Omron CX-Programmer project NewProject (CX-Programmer 9.75)

# PLC NewPLC1: CP2E-N N

## Global symbols (name address type ; comment)
W2.00 BOOL  ; ModbusStatus
0.00 BOOL  ; PROXY STOP KONVEYOR
0.01 BOOL  ; PROXY BOWL DISPENSER
0.02 BOOL  ; START BUTTON
100.00 BOOL  ; MOTOR BOWL DISPENSER
100.01 BOOL  ; MOTOR KONVEYOR
100.02 BOOL  ; MOTOR KONVEYOR
100.06 BOOL  ; MOTOR LINEAR ACTUATOR
10.02 BOOL  ; Cup Dispensed
200.00 BOOL  ; RELAY START
200.01 BOOL  ; RELAY START KONVEYOR
200.02 BOOL  ; RELAY ACTUATOR
200.03 BOOL  ; MOTOR BOWL
200.04 BOOL  ; RESET COUNTER
C0 CHANNEL  ; COMPILE MOTOR BOWL
T000 BOOL  ; TIMER ACTUATOR
T001 BOOL  ; TIMER START KONVEYOR
T002 BOOL  ; TIMER START KONVEYOR AFTER BOWL
T003 BOOL  ; START BOWL
W100.01 BOOL  ; MieKering_Ready
W100.02 BOOL  ; Cup_Jalan
W100.03 BOOL  ; RebusMie1_Start
W100.04 BOOL  ; RebusMie1_Done
W100.05 BOOL  ; RebusMie2_Start
W100.06 BOOL  ; RebusMie2_Done
W100.07 BOOL  ; RebusMie3_Start
W100.08 BOOL  ; RebusMie3_Done
W100.09 BOOL  ; Picked Cup
W10.00 BOOL  ; RST
W10.01 BOOL  ; MieKering_Picked
W10.02 BOOL  ; Cup dispensed
W10.03 BOOL  ; CupReady
W11.00 BOOL  ; Delay 1sec Trigger
W12.00 BOOL  ; 1 Sec Delay
W1.00 BOOL  ; MieKering_Arrived
W1.01 BOOL  ; MieKering_Picked
W1.02 BOOL  ; Cup_Dropped
W5.00 BOOL  ; Start MODBUS
FB_MODBUSTCP_SERVER _CP2E003_ExecuteModTcpServer
Order1_Menu D110 CHANNEL
Order1_Topping1 D100 CHANNEL
Order1_Topping2 D101 CHANNEL
Order1_Topping3 D102 CHANNEL
Order2_Menu D111 CHANNEL
Order2_Topping1 D103 CHANNEL
Order2_Topping2 D104 CHANNEL
Order2_Topping3 D105 CHANNEL
Order3_Menu D112 CHANNEL
Order3_Topping1 D106 CHANNEL
Order3_Topping2 D107 CHANNEL
Order3_Topping3 D108 CHANNEL
Start_Order W100.00 BOOL

## Program MODBUS (cyclic task 0)

### Section MODBUS

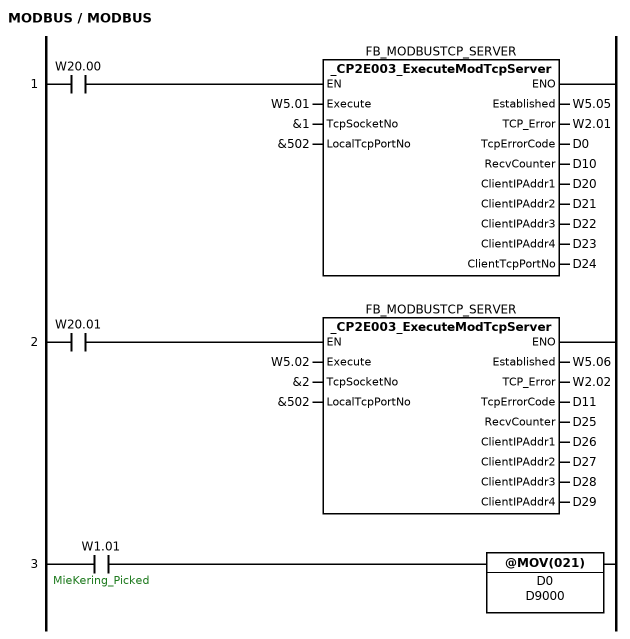
; rung 1
LD W20.00
CALL FB_MODBUSTCP_SERVER : _CP2E003_ExecuteModTcpServer (Execute := W5.01, TcpSocketNo := &1, LocalTcpPortNo := &502, Established => W5.05, TCP_Error => W2.01, TcpErrorCode => D0, RecvCounter => D10, ClientIPAddr1 => D20, ClientIPAddr2 => D21, ClientIPAddr3 => D22, ClientIPAddr4 => D23, ClientTcpPortNo => D24)
; rung 2
LD W20.01
CALL FB_MODBUSTCP_SERVER : _CP2E003_ExecuteModTcpServer (Execute := W5.02, TcpSocketNo := &2, LocalTcpPortNo := &502, Established => W5.06, TCP_Error => W2.02, TcpErrorCode => D11, RecvCounter => D25, ClientIPAddr1 => D26, ClientIPAddr2 => D27, ClientIPAddr3 => D28, ClientIPAddr4 => D29)
; rung 3
LD W1.01  ; MieKering_Picked
@MOV(021) D0 D9000

### Section Main

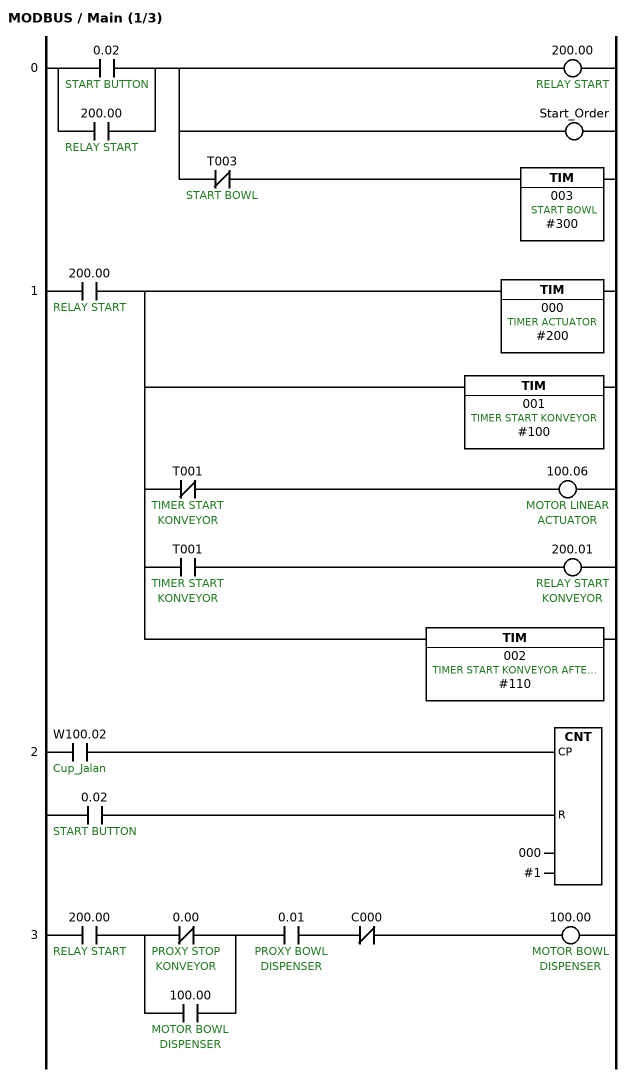
; rung 0
LD 0.02  ; START BUTTON
OR 200.00  ; RELAY START
OUT 200.00  ; RELAY START
OUT Start_Order
ANDNOT T003  ; START BOWL
TIM 003 #300  ; START BOWL
; rung 1
LD 200.00  ; RELAY START
OUT TR0
TIM 000 #200  ; TIMER ACTUATOR
TIM 001 #100  ; TIMER START KONVEYOR
ANDNOT T001  ; TIMER START KONVEYOR
OUT 100.06  ; MOTOR LINEAR ACTUATOR
LD TR0
AND T001  ; TIMER START KONVEYOR
OUT 200.01  ; RELAY START KONVEYOR
LD TR0
TIM 002 #110  ; TIMER START KONVEYOR AFTER BOWL
; rung 2
LD W100.02  ; Cup_Jalan
LD 0.02  ; START BUTTON
CNT 000 #1
; rung 3
LD 200.00  ; RELAY START
LDNOT 0.00  ; PROXY STOP KONVEYOR
OR 100.00  ; MOTOR BOWL DISPENSER
ANDLD
AND 0.01  ; PROXY BOWL DISPENSER
ANDNOT C000
OUT 100.00  ; MOTOR BOWL DISPENSER

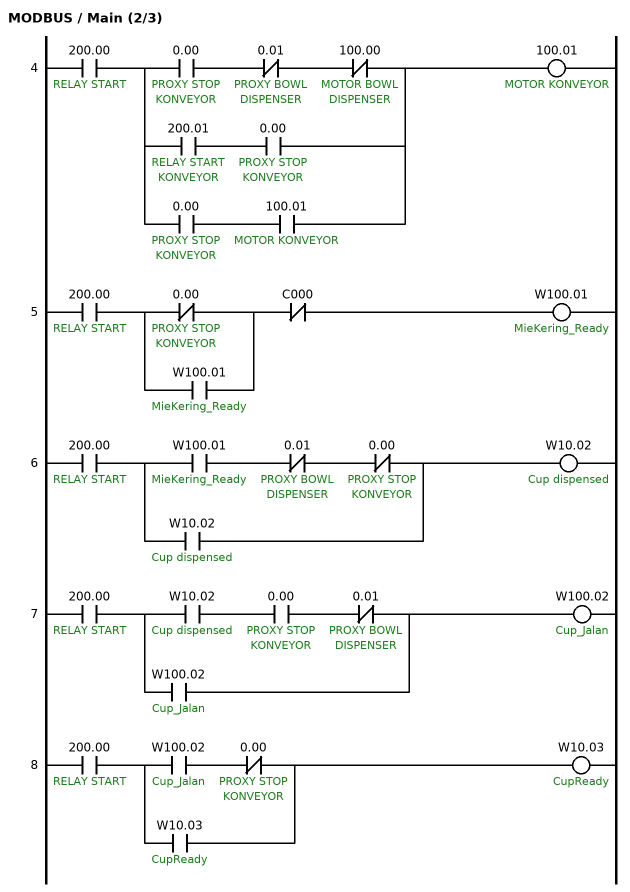
; rung 4
LD 200.00  ; RELAY START
LD 0.00  ; PROXY STOP KONVEYOR
ANDNOT 0.01  ; PROXY BOWL DISPENSER
ANDNOT 100.00  ; MOTOR BOWL DISPENSER
LD 200.01  ; RELAY START KONVEYOR
AND 0.00  ; PROXY STOP KONVEYOR
ORLD
LD 0.00  ; PROXY STOP KONVEYOR
AND 100.01  ; MOTOR KONVEYOR
ORLD
ANDLD
OUT 100.01  ; MOTOR KONVEYOR
; rung 5
LD 200.00  ; RELAY START
LDNOT 0.00  ; PROXY STOP KONVEYOR
OR W100.01  ; MieKering_Ready
ANDLD
ANDNOT C000
OUT W100.01  ; MieKering_Ready
; rung 6
LD 200.00  ; RELAY START
LD W100.01  ; MieKering_Ready
ANDNOT 0.01  ; PROXY BOWL DISPENSER
ANDNOT 0.00  ; PROXY STOP KONVEYOR
OR W10.02  ; Cup dispensed
ANDLD
OUT W10.02  ; Cup dispensed
; rung 7
LD 200.00  ; RELAY START
LD W10.02  ; Cup dispensed
AND 0.00  ; PROXY STOP KONVEYOR
ANDNOT 0.01  ; PROXY BOWL DISPENSER
OR W100.02  ; Cup_Jalan
ANDLD
OUT W100.02  ; Cup_Jalan
; rung 8
LD 200.00  ; RELAY START
LD W100.02  ; Cup_Jalan
ANDNOT 0.00  ; PROXY STOP KONVEYOR
OR W10.03  ; CupReady
ANDLD
OUT W10.03  ; CupReady

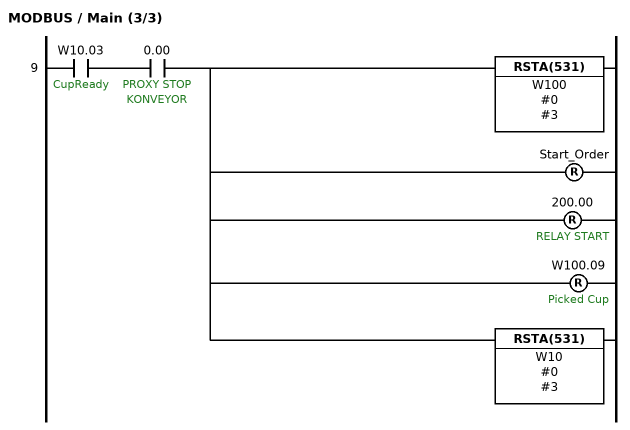
; rung 9
LD W10.03  ; CupReady
AND 0.00  ; PROXY STOP KONVEYOR
RSTA(531) W100 #0 #3
RSET Start_Order
RSET 200.00  ; RELAY START
RSET W100.09  ; Picked Cup
RSTA(531) W10 #0 #3

### Section Delay_Timer

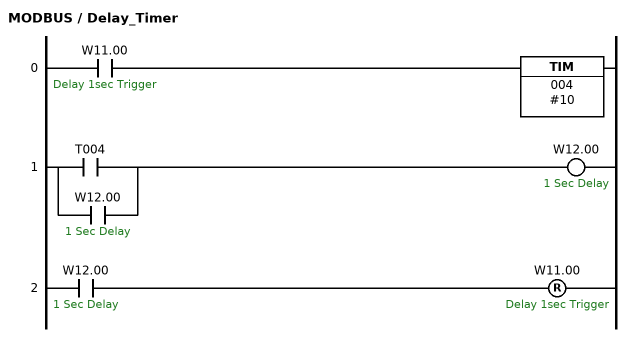
; rung 0
LD W11.00  ; Delay 1sec Trigger
TIM 004 #10
; rung 1
LD T004
OR W12.00  ; 1 Sec Delay
OUT W12.00  ; 1 Sec Delay
; rung 2
LD W12.00  ; 1 Sec Delay
RSET W11.00  ; Delay 1sec Trigger

### Section END
; rung 0
END(001)

## Function block _CP2E003_ExecuteModTcpServer (Omron library block, body left out)